// Mitsubishi GX Works2 project: 세척공정withAGV   PLC: Q02U

PROGRAM MAIN
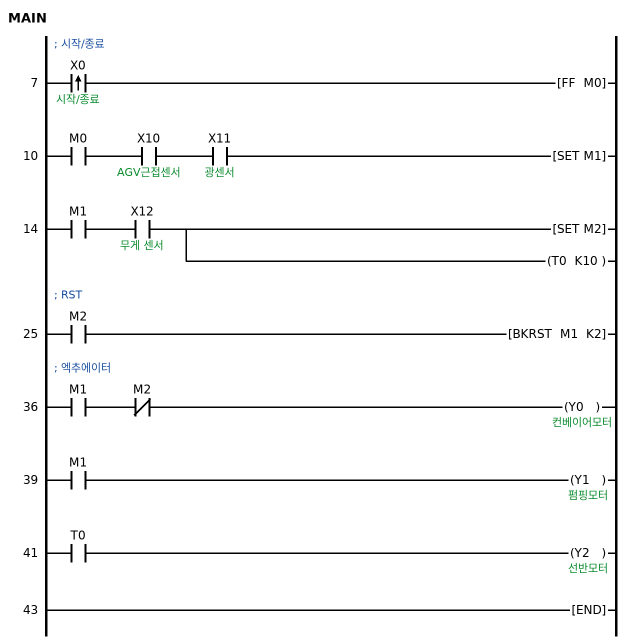
; 시작/종료
7     LDP     X0  ; 시작/종료
      FF      M0
10    LD      M0
      AND     X10  ; AGV근접센서
      AND     X11  ; 광센서
      SET     M1
14    LD      M1
      AND     X12  ; 무게 센서
      SET     M2
      OUT     T0 K10
; RST
25    LD      M2
      BKRST   M1 K2
; 엑추에이터
36    LD      M1
      ANI     M2
      OUT     Y0  ; 컨베이어모터
39    LD      M1
      OUT     Y1  ; 펌핑모터
41    LD      T0
      OUT     Y2  ; 선반모터
43    END
END_PROGRAM
